// TIA Portal V20 export
// export: Created 2025-12-01T14:57:13.1688662Z, ExportSetting None, DisplayName Totally Integrated Automation Portal, DisplayVersion V20 Update 3, DisplayName TIA Portal Openness, DisplayVersion V20 Update 3, DisplayName TIA Portal Version Control Interface, DisplayVersion V20 Update 3, DisplayName STEP 7 Professional, DisplayVersion V20 Update 3, DisplayName STEP 7 Safety, DisplayVersion V20 Update 2, DisplayName WinCC Basic/Comfort/Advanced, DisplayVersion V20 Update 3, DisplayName WinCC Professional, DisplayVersion V20 Update 3, DisplayName WinCC Unified, DisplayVersion V20 Update 3
FUNCTION "FC879_Transferir_GaliboDeUT" : Void   // FC879, LAD
{ S7_Optimized_Access := 'TRUE' }
// stored: AutoNumber false, SetENOAutomatically false
   VAR_INPUT
      Mesa : UInt;
      NumeroUT : UInt;
   END_VAR
BEGIN

NETWORK
TITLE = Distribuir >>> Del tipo de CODIGO del Galibo
/////////////////////////////////////////////////////////////////////////////
/// Dependiendo del CODIGO DE GALIBO >>> Se guarda Diferente
      SET;
      AN    "DB850_DefinicionMesas".Mesa[#Mesa].ConfigFB.Galibo;
      JC    CodigoAntiguo;
      JU    CodigoActual;



NETWORK
TITLE = CODIGO ANTIGUO >>> Transferir a la UT - Galibo
CodigoAntiguo:NOP   0;

/////////////////////////////////////////////////////////////////////////////
/////////////////////////////////////////////////////////////////////////////
/////////////////////////////////////////////////////////////////////////////
// --- GALIBO --> Remontado / Largura / Anchura / Altura


/////////////////////////////////////////////////////////////////////////////
// -- Codigo de Altura
      SET;  // Hay que guardar la altura ?
      AN    "DB850_DefinicionMesas".Mesa[#Mesa].AtributosGalibo_Guardar.Altura;
      JC    CodigoAntiguo_NoHay_CodigoAltura;

      L     "DB875_DatosGalibo".Galibo[#Mesa].Codigo.Galibo;
      AW    16#000F;
      T     "DB815_UTs_Datos".UT[#NumeroUT].GaliboAltura;

      L     "DB875_DatosGalibo".Galibo[#Mesa].GaliboVacia;
      T     "DB815_UTs_Datos".UT[#NumeroUT].GaliboVacia;

CodigoAntiguo_NoHay_CodigoAltura:NOP   0;


/////////////////////////////////////////////////////////////////////////////
// -- Codigo de Anchura
      SET;  // Hay que guardar la anchura ?
      AN    "DB850_DefinicionMesas".Mesa[#Mesa].AtributosGalibo_Guardar.Anchura;
      JC    CodigoAntiguo_NoHay_CodigoAnchura;

      L     "DB875_DatosGalibo".Galibo[#Mesa].Codigo.Galibo;
      AW    16#00F0;
      SRD   4;
      T     "DB815_UTs_Datos".UT[#NumeroUT].GaliboAnchura;

CodigoAntiguo_NoHay_CodigoAnchura:NOP   0;


/////////////////////////////////////////////////////////////////////////////
// -- Codigo de Largura
      SET;  // Hay que guardar la largura ?
      AN    "DB850_DefinicionMesas".Mesa[#Mesa].AtributosGalibo_Guardar.Profundidad;
      JC    CodigoAntiguo_NoHay_CodigoLargura;

      L     "DB875_DatosGalibo".Galibo[#Mesa].Codigo.Galibo;
      AW    16#0F00;
      SRD   8;
      T     "DB815_UTs_Datos".UT[#NumeroUT].GaliboProfundidad;

CodigoAntiguo_NoHay_CodigoLargura:NOP   0;


/////////////////////////////////////////////////////////////////////////////
// -- Codigo de Remontado
      SET;  // Hay que guardar la remontado ?
      AN    "DB850_DefinicionMesas".Mesa[#Mesa].AtributosGalibo_Guardar.Remontado;
      JC    CodigoAntiguo_NoHay_CodigoRemontado;

      L     "DB875_DatosGalibo".Galibo[#Mesa].Codigo.Galibo;
      AW    16#F000;
      SRD   12;
      T     "DB815_UTs_Datos".UT[#NumeroUT].GaliboRemontada;

CodigoAntiguo_NoHay_CodigoRemontado:NOP   0;



NETWORK
TITLE = CODIGO ANTIGUO >>> Transferir a la UT - Hueco Taco
/////////////////////////////////////////////////////////////////////////////
/////////////////////////////////////////////////////////////////////////////
/////////////////////////////////////////////////////////////////////////////
// --- HUECOTACO --> Tipo Carga / Hueco R / Hueco / Taco


/////////////////////////////////////////////////////////////////////////////
// -- Codigo de Taco
      SET;  // Hay que guardar la taco ?
      AN    "DB850_DefinicionMesas".Mesa[#Mesa].AtributosGalibo_Guardar.Taco;
      JC    CodigoAntiguo_NoHay_CodigoTaco;

      L     "DB875_DatosGalibo".Galibo[#Mesa].Codigo.HuecoTaco;
      AW    16#000F;
      T     "DB815_UTs_Datos".UT[#NumeroUT].GaliboTaco;

CodigoAntiguo_NoHay_CodigoTaco:NOP   0;


/////////////////////////////////////////////////////////////////////////////
// -- Codigo de Hueco
      SET;  // Hay que guardar la hueco ?
      AN    "DB850_DefinicionMesas".Mesa[#Mesa].AtributosGalibo_Guardar.Hueco;
      JC    CodigoAntiguo_NoHay_CodigoHueco;

      L     "DB875_DatosGalibo".Galibo[#Mesa].Codigo.HuecoTaco;
      AW    16#00F0;
      SRD   4;
      T     "DB815_UTs_Datos".UT[#NumeroUT].GaliboHueco;

CodigoAntiguo_NoHay_CodigoHueco:NOP   0;


/////////////////////////////////////////////////////////////////////////////
// -- Codigo de Hueco De Remontado
      SET;  // Hay que guardar la hueco R. ?
      AN    "DB850_DefinicionMesas".Mesa[#Mesa].AtributosGalibo_Guardar.HuecoRemontado;
      JC    CodigoAntiguo_NoHay_CodigoHuecoDeRemontado;

      L     "DB875_DatosGalibo".Galibo[#Mesa].Codigo.HuecoTaco;
      AW    16#0F00;
      SRD   8;
      T     "DB815_UTs_Datos".UT[#NumeroUT].GaliboHuecoRemontado;

CodigoAntiguo_NoHay_CodigoHuecoDeRemontado:NOP   0;


/////////////////////////////////////////////////////////////////////////////
// -- Codigo de Tipo de Carga
      SET;  // Hay que guardar la tipo carga ?
      AN    "DB850_DefinicionMesas".Mesa[#Mesa].AtributosGalibo_Guardar.Tipo;
      JC    CodigoAntiguo_NoHay_CodigoTipoDeCarga;

      L     "DB875_DatosGalibo".Galibo[#Mesa].Codigo.HuecoTaco;
      AW    16#F000;
      SRD   12;
      T     "DB815_UTs_Datos".UT[#NumeroUT].GaliboTipoCarga;

CodigoAntiguo_NoHay_CodigoTipoDeCarga:NOP   0;



NETWORK
TITLE = CODIGO ANTIGUO >>> Transferir a la UT - Galibo Extra
/////////////////////////////////////////////////////////////////////////////
/////////////////////////////////////////////////////////////////////////////
/////////////////////////////////////////////////////////////////////////////
// --- GALIBOEXTRA --> ???? / ???? / ???? / Color


/////////////////////////////////////////////////////////////////////////////
// -- Codigo de Color
      SET;  // Hay que guardar el color ?
      AN    "DB850_DefinicionMesas".Mesa[#Mesa].AtributosGalibo_Guardar.Color;
      JC    CodigoAntiguo_NoHay_CodigoColor;

      L     "DB875_DatosGalibo".Galibo[#Mesa].Codigo.GaliboExtra;
      AW    16#000F;
      T     "DB815_UTs_Datos".UT[#NumeroUT].GaliboColor;

CodigoAntiguo_NoHay_CodigoColor:NOP   0;


/////////////////////////////////////////////////////////////////////////////
// -- Codigo de Patin
      SET;  // Hay que guardar Patin
      AN    "DB850_DefinicionMesas".Mesa[#Mesa].AtributosGalibo_Guardar.Patin;
      JC    CodigoAntiguo_NoHay_CodigoPatin;

      L     "DB875_DatosGalibo".Galibo[#Mesa].Codigo.GaliboExtra;
      AW    16#00F0;
      SRD   4;
      T     "DB815_UTs_Datos".UT[#NumeroUT].GaliboPatin;

CodigoAntiguo_NoHay_CodigoPatin:NOP   0;



NETWORK
TITLE = CODIGO ANTIGUO >>> Transferir a la UT - Cota de Altura
/////////////////////////////////////////////////////////////////////////////
/////////////////////////////////////////////////////////////////////////////
/////////////////////////////////////////////////////////////////////////////
// --- COTA DE ALTURA
      SET;
      AN    "DB850_DefinicionMesas".Mesa[#Mesa].AtributosGalibo_Guardar.Cota_Altura;
      JC    CodigoAntiguo_NoHay_CotaAltura;

      L     "DB875_DatosGalibo".Galibo[#Mesa].CotaAltura;
      T     "DB815_UTs_Datos".UT[#NumeroUT].CotaAltura;

CodigoAntiguo_NoHay_CotaAltura:NOP   0;



NETWORK
TITLE = CODIGO ANTIGUO >>> Transferir a la UT - Cota de Anchura
/////////////////////////////////////////////////////////////////////////////
/////////////////////////////////////////////////////////////////////////////
/////////////////////////////////////////////////////////////////////////////
// --- COTA DE ANCHURA
      SET;
      AN    "DB850_DefinicionMesas".Mesa[#Mesa].AtributosGalibo_Guardar.Cota_Anchura;
      JC    CodigoAntiguo_NoHay_CotaAnchura;

      L     "DB875_DatosGalibo".Galibo[#Mesa].CotaAnchura;
      T     "DB815_UTs_Datos".UT[#NumeroUT].CotaAnchura;

CodigoAntiguo_NoHay_CotaAnchura:NOP   0;



NETWORK
TITLE = CODIGO ANTIGUO >>> Transferir a la UT - Cota de Largura
/////////////////////////////////////////////////////////////////////////////
/////////////////////////////////////////////////////////////////////////////
/////////////////////////////////////////////////////////////////////////////
// --- COTA DE LARGURA
      SET;
      AN    "DB850_DefinicionMesas".Mesa[#Mesa].AtributosGalibo_Guardar.Cota_Profundidad;
      JC    CodigoAntiguo_NoHay_CotaLargura;

      L     "DB875_DatosGalibo".Galibo[#Mesa].CotaProfundidad;
      T     "DB815_UTs_Datos".UT[#NumeroUT].CotaProfundidad;

CodigoAntiguo_NoHay_CotaLargura:NOP   0;



NETWORK
TITLE = CODIGO ANTIGUO >>> Transferir a la UT - Peso
/////////////////////////////////////////////////////////////////////////////
/////////////////////////////////////////////////////////////////////////////
/////////////////////////////////////////////////////////////////////////////
// ---  PESO
      SET;
      AN    "DB850_DefinicionMesas".Mesa[#Mesa].AtributosGalibo_Guardar.Peso;
      JC    CodigoAntiguo_NoHay_Peso;

      L     "DB875_DatosGalibo".Galibo[#Mesa].Peso;
      T     "DB815_UTs_Datos".UT[#NumeroUT].Peso;

CodigoAntiguo_NoHay_Peso:NOP   0;



NETWORK
TITLE = CODIGO ANTIGUO >>> Transferir a la UT - Etiqueta Router
/////////////////////////////////////////////////////////////////////////////
/////////////////////////////////////////////////////////////////////////////
/////////////////////////////////////////////////////////////////////////////
// ---  ETIQUETA de Router
      SET;
      AN    "DB850_DefinicionMesas".Mesa[#Mesa].AtributosGalibo_Guardar.EtiquetaRouter;
      JC    CodigoAntiguo_NoHay_EtiquetaRouter;

      L     "DB875_DatosGalibo".Galibo[#Mesa].EtiquetaRouter;
      T     "DB814_UTs_Etiqueta".UT[#NumeroUT].EtiquetaRouter;

CodigoAntiguo_NoHay_EtiquetaRouter:NOP   0;



NETWORK
TITLE = CODIGO ANTIGUO >>> Final
/////////////////////////////////////////////////////////////////////////////
/////////////////////////////////////////////////////////////////////////////
/////////////////////////////////////////////////////////////////////////////
// ---  FINAL
      BE;



NETWORK
TITLE = CODIGO ACTUAL 2023 >>> Transferir a la UT - Galibo
CodigoActual:NOP   0;

/////////////////////////////////////////////////////////////////////////////
/////////////////////////////////////////////////////////////////////////////
/////////////////////////////////////////////////////////////////////////////
// --- GALIBO --> Remontado / Largura / Anchura / Altura


/////////////////////////////////////////////////////////////////////////////
// -- Codigo de Altura
      SET;  // Hay que guardar la altura ?
      AN    "DB850_DefinicionMesas".Mesa[#Mesa].AtributosGalibo_Guardar.Altura;
      JC    CodigoActual_NoHay_CodigoAltura;

      L     "DB875_DatosGalibo".Galibo[#Mesa].GaliboAltura;
      T     "DB815_UTs_Datos".UT[#NumeroUT].GaliboAltura;

      L     "DB875_DatosGalibo".Galibo[#Mesa].GaliboVacia;
      T     "DB815_UTs_Datos".UT[#NumeroUT].GaliboVacia;


CodigoActual_NoHay_CodigoAltura:NOP   0;


/////////////////////////////////////////////////////////////////////////////
// -- Codigo de Anchura
      SET;  // Hay que guardar la anchura ?
      AN    "DB850_DefinicionMesas".Mesa[#Mesa].AtributosGalibo_Guardar.Anchura;
      JC    CodigoActual_NoHay_CodigoAnchura;

      L     "DB875_DatosGalibo".Galibo[#Mesa].GaliboAnchura;
      T     "DB815_UTs_Datos".UT[#NumeroUT].GaliboAnchura;

CodigoActual_NoHay_CodigoAnchura:NOP   0;


/////////////////////////////////////////////////////////////////////////////
// -- Codigo de Largura
      SET;  // Hay que guardar la largura ?
      AN    "DB850_DefinicionMesas".Mesa[#Mesa].AtributosGalibo_Guardar.Profundidad;
      JC    CodigoActual_NoHay_CodigoLargura;

      L     "DB875_DatosGalibo".Galibo[#Mesa].GaliboProfundidad;
      T     "DB815_UTs_Datos".UT[#NumeroUT].GaliboProfundidad;

CodigoActual_NoHay_CodigoLargura:NOP   0;


/////////////////////////////////////////////////////////////////////////////
// -- Codigo de Remontado
      SET;  // Hay que guardar la remontado ?
      AN    "DB850_DefinicionMesas".Mesa[#Mesa].AtributosGalibo_Guardar.Remontado;
      JC    CodigoActual_NoHay_CodigoRemontado;

      L     "DB875_DatosGalibo".Galibo[#Mesa].GaliboRemontada;
      T     "DB815_UTs_Datos".UT[#NumeroUT].GaliboRemontada;

CodigoActual_NoHay_CodigoRemontado:NOP   0;



NETWORK
TITLE = CODIGO ACTUAL 2023 >>> Transferir a la UT - Hueco Taco
/////////////////////////////////////////////////////////////////////////////
/////////////////////////////////////////////////////////////////////////////
/////////////////////////////////////////////////////////////////////////////
// --- HUECOTACO --> Tipo Carga / Hueco R / Hueco / Taco


/////////////////////////////////////////////////////////////////////////////
// -- Codigo de Taco
      SET;  // Hay que guardar la taco ?
      AN    "DB850_DefinicionMesas".Mesa[#Mesa].AtributosGalibo_Guardar.Taco;
      JC    CodigoActual_NoHay_CodigoTaco;

      L     "DB875_DatosGalibo".Galibo[#Mesa].GaliboTaco;
      T     "DB815_UTs_Datos".UT[#NumeroUT].GaliboTaco;

CodigoActual_NoHay_CodigoTaco:NOP   0;


/////////////////////////////////////////////////////////////////////////////
// -- Codigo de Hueco
      SET;  // Hay que guardar la hueco ?
      AN    "DB850_DefinicionMesas".Mesa[#Mesa].AtributosGalibo_Guardar.Hueco;
      JC    CodigoActual_NoHay_CodigoHueco;

      L     "DB875_DatosGalibo".Galibo[#Mesa].GaliboHueco;
      T     "DB815_UTs_Datos".UT[#NumeroUT].GaliboHueco;

CodigoActual_NoHay_CodigoHueco:NOP   0;


/////////////////////////////////////////////////////////////////////////////
// -- Codigo de Hueco De Remontado
      SET;  // Hay que guardar la hueco R. ?
      AN    "DB850_DefinicionMesas".Mesa[#Mesa].AtributosGalibo_Guardar.HuecoRemontado;
      JC    CodigoActual_NoHay_CodigoHuecoDeRemontado;

      L     "DB875_DatosGalibo".Galibo[#Mesa].GaliboHuecoRemontado;
      T     "DB815_UTs_Datos".UT[#NumeroUT].GaliboHuecoRemontado;

CodigoActual_NoHay_CodigoHuecoDeRemontado:NOP   0;


/////////////////////////////////////////////////////////////////////////////
// -- Codigo de Tipo de Carga
      SET;  // Hay que guardar la tipo carga ?
      AN    "DB850_DefinicionMesas".Mesa[#Mesa].AtributosGalibo_Guardar.Tipo;
      JC    CodigoActual_NoHay_CodigoTipoDeCarga;

      L     "DB875_DatosGalibo".Galibo[#Mesa].GaliboTipoCarga;
      T     "DB815_UTs_Datos".UT[#NumeroUT].GaliboTipoCarga;

CodigoActual_NoHay_CodigoTipoDeCarga:NOP   0;



NETWORK
TITLE = CODIGO ACTUAL 2023 >>> Transferir a la UT - Galibo Extra
/////////////////////////////////////////////////////////////////////////////
/////////////////////////////////////////////////////////////////////////////
/////////////////////////////////////////////////////////////////////////////
// --- GALIBOEXTRA --> ???? / ???? / ???? / Color


/////////////////////////////////////////////////////////////////////////////
// -- Codigo de Color
      SET;  // Hay que guardar el color ?
      AN    "DB850_DefinicionMesas".Mesa[#Mesa].AtributosGalibo_Guardar.Color;
      JC    CodigoActual_NoHay_CodigoColor;

      L     "DB875_DatosGalibo".Galibo[#Mesa].GaliboColor;
      T     "DB815_UTs_Datos".UT[#NumeroUT].GaliboColor;

CodigoActual_NoHay_CodigoColor:NOP   0;


/////////////////////////////////////////////////////////////////////////////
// -- Codigo de Patin
      SET;  // Hay que guardar Patin
      AN    "DB850_DefinicionMesas".Mesa[#Mesa].AtributosGalibo_Guardar.Patin;
      JC    CodigoActual_NoHay_CodigoPatin;

      L     "DB875_DatosGalibo".Galibo[#Mesa].GaliboPatin;
      T     "DB815_UTs_Datos".UT[#NumeroUT].GaliboPatin;

CodigoActual_NoHay_CodigoPatin:NOP   0;



NETWORK
TITLE = CODIGO ACTUAL 2023 >>> Transferir a la UT - Cota de Altura
/////////////////////////////////////////////////////////////////////////////
/////////////////////////////////////////////////////////////////////////////
/////////////////////////////////////////////////////////////////////////////
// --- COTA DE ALTURA
      SET;
      AN    "DB850_DefinicionMesas".Mesa[#Mesa].AtributosGalibo_Guardar.Cota_Altura;
      JC    CodigoActual_NoHay_CotaAltura;

      L     "DB875_DatosGalibo".Galibo[#Mesa].CotaAltura;
      T     "DB815_UTs_Datos".UT[#NumeroUT].CotaAltura;

CodigoActual_NoHay_CotaAltura:NOP   0;



NETWORK
TITLE = CODIGO ACTUAL 2023 >>> Transferir a la UT - Cota de Anchura
/////////////////////////////////////////////////////////////////////////////
/////////////////////////////////////////////////////////////////////////////
/////////////////////////////////////////////////////////////////////////////
// --- COTA DE ANCHURA
      SET;
      AN    "DB850_DefinicionMesas".Mesa[#Mesa].AtributosGalibo_Guardar.Cota_Anchura;
      JC    CodigoActual_NoHay_CotaAnchura;

      L     "DB875_DatosGalibo".Galibo[#Mesa].CotaAnchura;
      T     "DB815_UTs_Datos".UT[#NumeroUT].CotaAnchura;

CodigoActual_NoHay_CotaAnchura:NOP   0;



NETWORK
TITLE = CODIGO ACTUAL 2023 >>> Transferir a la UT - Cota de Largura
/////////////////////////////////////////////////////////////////////////////
/////////////////////////////////////////////////////////////////////////////
/////////////////////////////////////////////////////////////////////////////
// --- COTA DE LARGURA
      SET;
      AN    "DB850_DefinicionMesas".Mesa[#Mesa].AtributosGalibo_Guardar.Cota_Profundidad;
      JC    CodigoActual_NoHay_CotaLargura;

      L     "DB875_DatosGalibo".Galibo[#Mesa].CotaProfundidad;
      T     "DB815_UTs_Datos".UT[#NumeroUT].CotaProfundidad;

CodigoActual_NoHay_CotaLargura:NOP   0;



NETWORK
TITLE = CODIGO ACTUAL 2023 >>> Transferir a la UT - Peso
/////////////////////////////////////////////////////////////////////////////
/////////////////////////////////////////////////////////////////////////////
/////////////////////////////////////////////////////////////////////////////
// ---  PESO
      SET;
      AN    "DB850_DefinicionMesas".Mesa[#Mesa].AtributosGalibo_Guardar.Peso;
      JC    CodigoActual_NoHay_Peso;

      L     "DB875_DatosGalibo".Galibo[#Mesa].Peso;
      T     "DB815_UTs_Datos".UT[#NumeroUT].Peso;

CodigoActual_NoHay_Peso:NOP   0;



NETWORK
TITLE = CODIGO ACTUAL 2023 >>> Transferir a la UT - Etiqueta Router
/////////////////////////////////////////////////////////////////////////////
/////////////////////////////////////////////////////////////////////////////
/////////////////////////////////////////////////////////////////////////////
// ---  ETIQUETA de Router
      SET;
      AN    "DB850_DefinicionMesas".Mesa[#Mesa].AtributosGalibo_Guardar.EtiquetaRouter;
      JC    CodigoActual_NoHay_EtiquetaRouter;

      L     "DB875_DatosGalibo".Galibo[#Mesa].EtiquetaRouter;
      T     "DB814_UTs_Etiqueta".UT[#NumeroUT].EtiquetaRouter;

CodigoActual_NoHay_EtiquetaRouter:NOP   0;



NETWORK
TITLE = CODIGO ACTUAL 2023 >>> Final
/////////////////////////////////////////////////////////////////////////////
/////////////////////////////////////////////////////////////////////////////
/////////////////////////////////////////////////////////////////////////////
// ---  FINAL
      BE;


END_FUNCTION
